(* Logix 5000 project; controller PLC2_Project_5 Emulate 5570 rev 20.11; software revision 20.00 *)

TASK MainTask (continuous, watchdog 500 ms) : MainProgram

MODULES
   Local : Emulate 5570 (ICP 1, rev 20.11)
END_MODULES

PROGRAM MainProgram   (* main routine MainRoutine *)
VAR
   in_rotameterBit : BOOL; {access Read Only}
   Oil_TempTimerValue : REAL; {access Read Only}
   RefreshRate : TIMER := (PRE := 10000); {access Read Only}   // Calculation time / sample time
   RefreshRateSeconds : REAL; {access Read Only}
   Rotameter_gpm_1 : REAL; {access Read Only}
   Rotameter_gpm_2 : REAL; {access Read Only}
   Rotameter_gps_1 : REAL; {access Read Only}
   Rotameter_gps_2 : REAL; {access Read Only}
   Rotameter_In : BOOL; {access Read Only}
   Rotameter_K_Factor : REAL; {access Read Only}
   Rotameter_PulseCounter : COUNTER; {access Read Only}
   Rotameter_Pulses : COUNTER := (PRE := 9999); {access Read Only}
   Rotameter_TimeSinceLastPulse : TIMER := (PRE := 999999); {access Read Only}
   sim_rotameter : TIMER := (PRE := 5000);
   TempCalc : REAL; {access Read Only}
END_VAR

ROUTINE Input_Output   (* ladder *)
// Digital Input & Output
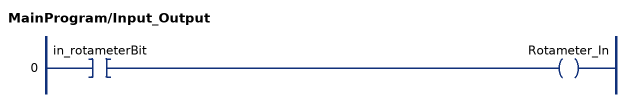
   0: XIC(in_rotameterBit)OTE(Rotameter_In);
END_ROUTINE

ROUTINE MainRoutine   (* ladder *)
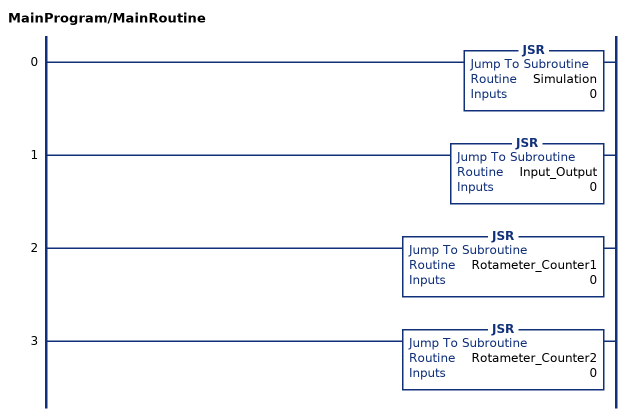
   0: JSR(Simulation,0);
   1: JSR(Input_Output,0);
   2: JSR(Rotameter_Counter1,0);
   3: JSR(Rotameter_Counter2,0);
END_ROUTINE

ROUTINE Rotameter_Counter1   (* ladder *)
// Measures the time between pulses in ms. Less reliable at higher pulse rates
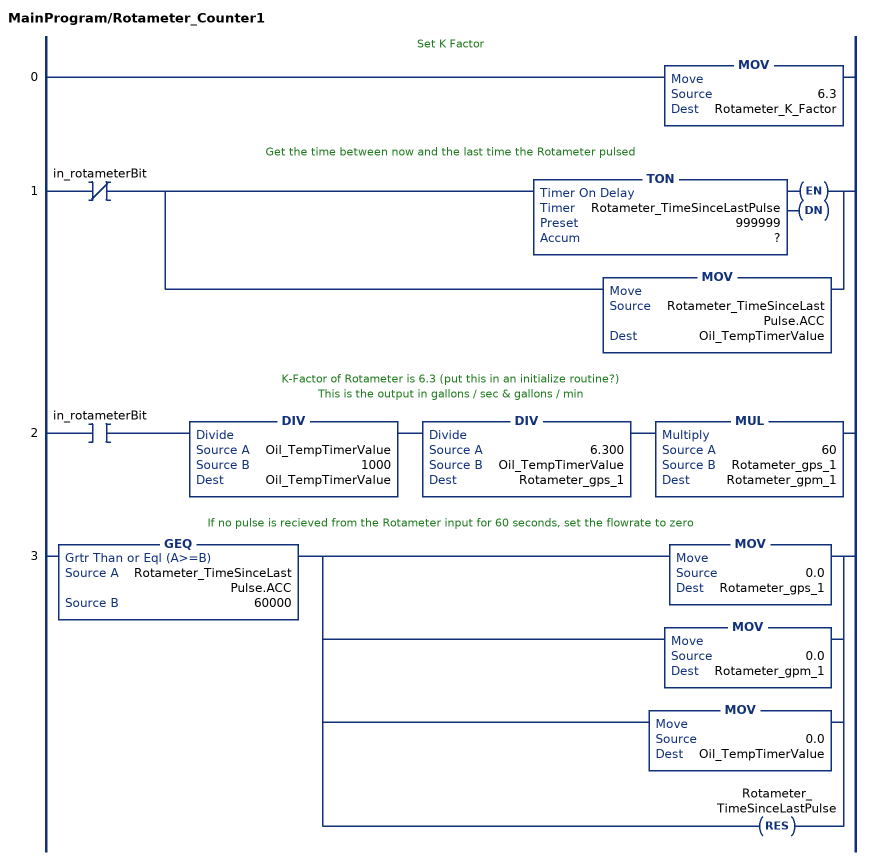
   // Set K Factor
   0: MOV(6.3,Rotameter_K_Factor);
   // Get the time between now and the last time the Rotameter pulsed
   1: XIO(in_rotameterBit)[TON(Rotameter_TimeSinceLastPulse,?,?) ,MOV(Rotameter_TimeSinceLastPulse.ACC,Oil_TempTimerValue) ];
   // K-Factor of Rotameter is 6.3 (put this in an initialize routine?)
   // This is the output in gallons / sec & gallons / min
   2: XIC(in_rotameterBit)DIV(Oil_TempTimerValue,1000,Oil_TempTimerValue)DIV(6.300,Oil_TempTimerValue,Rotameter_gps_1)MUL(60,Rotameter_gps_1,Rotameter_gpm_1);
   // If no pulse is recieved from the Rotameter input for 60 seconds, set the flowrate to zero
   3: GEQ(Rotameter_TimeSinceLastPulse.ACC,60000)[MOV(0.0,Rotameter_gps_1) ,MOV(0.0,Rotameter_gpm_1) ,MOV(0.0,Oil_TempTimerValue) ,RES(Rotameter_TimeSinceLastPulse) ];
END_ROUTINE

ROUTINE Rotameter_Counter2   (* ladder *)
// Measures the number of pulses within a set time interval. More reliable than counter1, but still becomes unstable at higher pulse frequencies
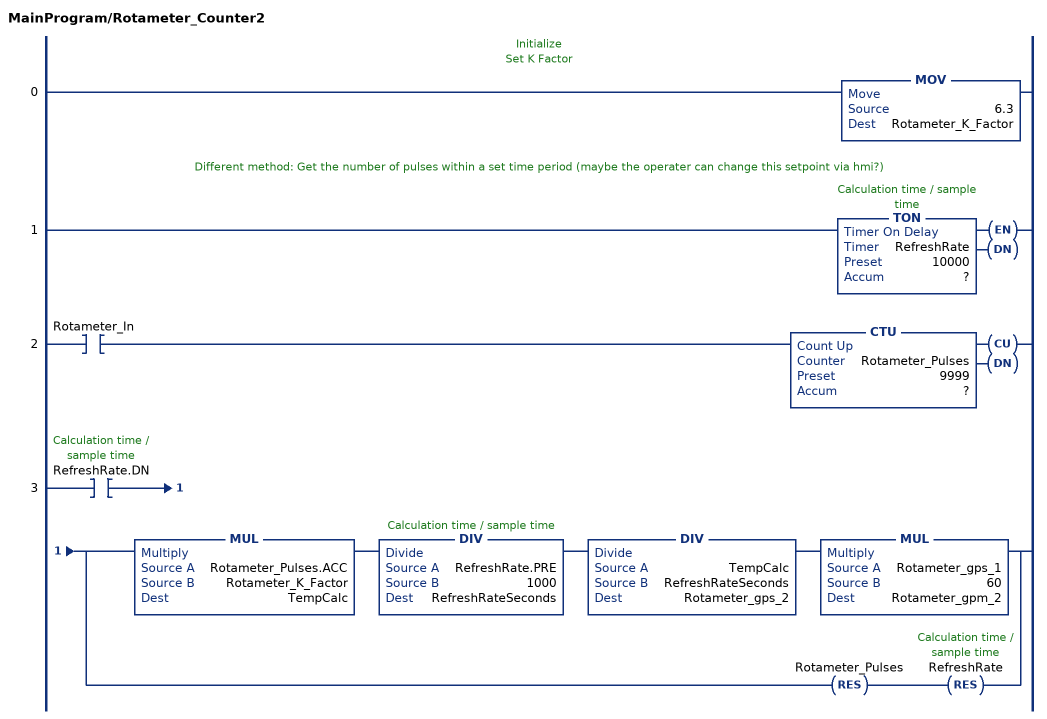
   // Initialize
   // Set K Factor
   0: MOV(6.3,Rotameter_K_Factor);
   // Different method: Get the number of pulses within a set time period (maybe the operater can change this setpoint via hmi?)
   1: TON(RefreshRate,?,?);
   2: XIC(Rotameter_In)CTU(Rotameter_Pulses,?,?);
   3: XIC(RefreshRate.DN)[MUL(Rotameter_Pulses.ACC,Rotameter_K_Factor,TempCalc) DIV(RefreshRate.PRE,1000,RefreshRateSeconds) DIV(TempCalc,RefreshRateSeconds,Rotameter_gps_2) MUL(Rotameter_gps_1,60,Rotameter_gpm_2) ,RES(Rotameter_Pulses) RES(RefreshRate) ];
END_ROUTINE

ROUTINE Simulation   (* ladder *)
// Simulates a rotameter input
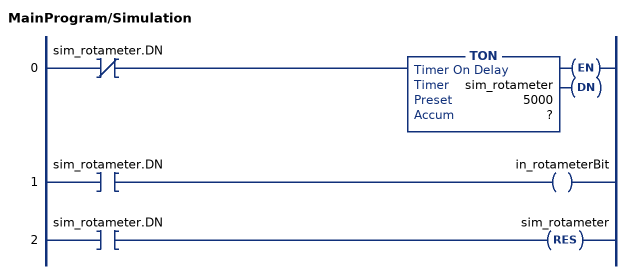
   0: XIO(sim_rotameter.DN)TON(sim_rotameter,?,?);
   1: XIC(sim_rotameter.DN)OTE(in_rotameterBit);
   2: XIC(sim_rotameter.DN)RES(sim_rotameter);
END_ROUTINE
END_PROGRAM
